{attribute 'GeneratedUsingTerminal: EL6201-0000-0017'}
{attribute addProperty BoxType "EL6201-0000-0017"}
{attribute addProperty Id "Slave_25A_DO0BOOL1Slave_25A_DO1BOOL1Slave_25A_DO2BOOL1Slave_25A_DO3BOOL1Slave_25B_DO0BOOL1Slave_25B_DO1BOOL1Slave_25B_DO2BOOL1Slave_25B_DO3BOOL1"}
{attribute addProperty CRC "156408758"}
{attribute addProperty Size "8"}
TYPE Slave_25_Outputs_09529BB6 :
STRUCT
	{attribute addProperty Name "Slave_25A_DO0"}
	Slave_25A_DO0 : BOOL;
	{attribute addProperty Name "Slave_25A_DO1"}
	Slave_25A_DO1 : BOOL;
	{attribute addProperty Name "Slave_25A_DO2"}
	Slave_25A_DO2 : BOOL;
	{attribute addProperty Name "Slave_25A_DO3"}
	Slave_25A_DO3 : BOOL;
	{attribute addProperty Name "Slave_25B_DO0"}
	Slave_25B_DO0 : BOOL;
	{attribute addProperty Name "Slave_25B_DO1"}
	Slave_25B_DO1 : BOOL;
	{attribute addProperty Name "Slave_25B_DO2"}
	Slave_25B_DO2 : BOOL;
	{attribute addProperty Name "Slave_25B_DO3"}
	Slave_25B_DO3 : BOOL;
END_STRUCT
END_TYPE

(* stored: Version 1.2.0.0, ProductVersion 3.1.4024.9
   DUT Slave_25_Outputs_09529BB6: Id {ac212217-751b-4ff8-be0d-0f64accff4a3} *)
